FUNCTION_BLOCK T_CommandInvoker EXTENDS T_NamedBase IMPLEMENTS I_CommandInvoker
VAR
  _commandQueue : I_CommandQueue;
  currentCmd : I_Task;
  
  state, prevState : (IDLE_STATE, GET_COMMAND, PROCESSING_STATE, ERROR_STATE) := IDLE_STATE;
  initialised : BOOL;
END_VAR

METHOD PUBLIC CyclicLogic
IF NOT initialised THEN
  RETURN;
END_IF

StateMachine();
END_METHOD

PROPERTY PUBLIC Error : BOOL
GET
Error := (STATE = ERROR_STATE);
END_GET
END_PROPERTY

PROPERTY PUBLIC Idle : BOOL
GET
Idle := (STATE = IDLE_STATE);
END_GET
END_PROPERTY

METHOD PUBLIC Initialise : BOOL
VAR_INPUT
  commandQueue : I_CommandQueue;
END_VAR
IF commandQueue = 0 THEN
  LogError('command queue = 0');
  RETURN;
END_IF

LogInfo('command queue initlaised');
_commandQueue := commandQueue;

initialised := TRUE;
Initialise := TRUE;
END_METHOD

PROPERTY PUBLIC Processing : BOOL
GET
Processing := (state = PROCESSING_STATE OR STATE = GET_COMMAND);
END_GET
END_PROPERTY

METHOD PUBLIC Reset
state := IDLE_STATE;
_commandQueue.Clear();
currentCmd := 0;
END_METHOD

METHOD PRIVATE StateChanged : BOOL
IF  state = prevState THEN
  RETURN;
END_IF

prevState := state;
StateChanged := TRUE;
END_METHOD

METHOD PRIVATE StateMachine
IF currentCmd <> 0 THEN
  currentCmd.CyclicLogic();
END_IF

CASE state OF
  IDLE_STATE:
    stateChanged();

    IF _commandQueue.Count > 0 THEN
      state := GET_COMMAND;
    END_IF

  GET_COMMAND:
    StateChanged();

    IF _commandQueue.GetNext(output_command => currentCmd) THEN
      state := PROCESSING_STATE;
    END_IF

  PROCESSING_STATE:

    IF StateChanged() THEN
      
      IF currentCmd = 0 THEN
        LogError('Command invoker target task is null');
        state := ERROR_STATE;
        RETURN;

      ELSE
        currentCmd.Execute();

      END_IF
      
    ELSIF currentCmd.Done THEN
      state := IDLE_STATE;
      
    END_IF

  ERROR_STATE:
    StateChanged();

END_CASE
END_METHOD

END_FUNCTION_BLOCK

(* stored: Version 1.1.0.1
   POU T_CommandInvoker: Id {284490e9-a282-4ae0-81ff-39283e67a745}, SpecialFunc None
   Folder Methods: Id {e521ab56-6a39-4e10-8f58-248d18c7733e}
   Folder Private: Id {2ca2c215-25a1-4974-b75f-8afbdd614f02}
   Folder Properties: Id {81f156f7-0e1d-4352-9c9d-91f3c14e4d7e}
   Method CyclicLogic: Id {613cd9fa-2eab-4fed-a024-e26149687420}
   Property Error: Id {145f7fdc-d96e-4b87-a7f8-91e7a5281c3e}
   Get Get: Id {1a47327a-80f2-4894-8f0e-71b28bafcdf3}
   Property Idle: Id {5162eb79-5a24-416b-9660-b17fe1883dd7}
   Get Get: Id {17d3595b-787e-4817-8ba8-e93080effbeb}
   Method Initialise: Id {922e36fe-7e8a-4a61-ae4b-07f4e809c5a0}
   Property Processing: Id {aa929904-bc0a-4138-a56c-b562d67de825}
   Get Get: Id {5ebb08e6-ddf8-463c-91a5-5e95949e148a}
   Method Reset: Id {5dccd8c1-7a08-4893-a164-e735d9c7e783}
   Method StateChanged: Id {e323c704-c3bd-4d64-aea1-b13b203bb45e}
   Method StateMachine: Id {47b697f6-4b7e-4114-9989-224ef356624a} *)
